Universal Robots PolyScope program: definitivo2.urp

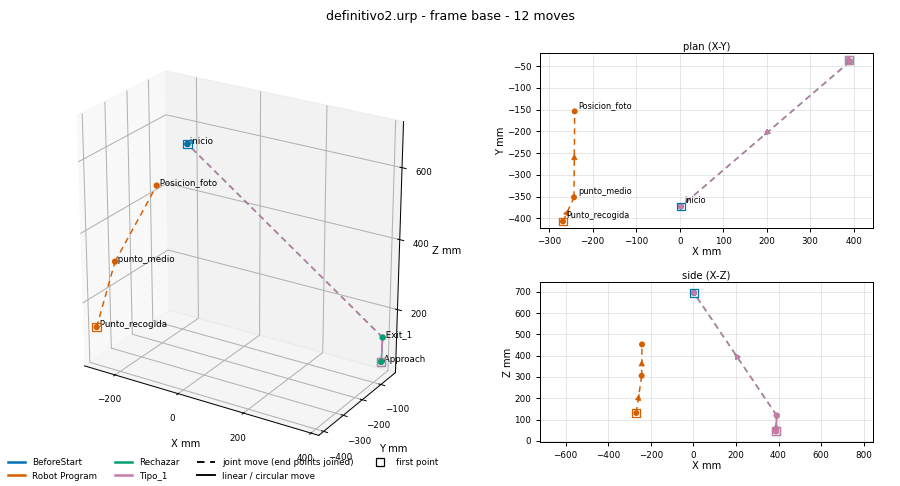
[picture p0: tool path of definitivo2.urp in frame base, 12 of 12 moves have a stored position in this frame; points joined in program order, loops and branches not executed]
Program definitivo2 (installation=default directory=/programs createdIn=5.14.5 lastSavedIn=5.14.5 robotSerialNumber=20195300809)
Calibrated DH parameters: a=[-0.000085, -0.20076, -0.212369, 0.000121, -0.000118, 0]; d=[0.15185, -26.306375, 24.753047, 1.684739, 0.085386, 0.092088]; alpha=[1.572149, -0.00522, -0.011864, 1.571339, -1.571085, 0]; deltaTheta=[0, 0.599885, -0.513355, -0.086555, 0.000006, 0]
InitVariablesNode variables(variable(name=Pallet_1_cnt_2, expression=1), variable(name=Pallet_1_cnt_3, expression=1), variable(name=Pallet_1_lct, expression=1), variable(name=Pallet_1_lct_1, expression=1), variable(name=Pallet_1_lno, expression=1), variable(name=Pallet_1_lno_1, expression=1), variable(name=Pallet_1_sep, expression=False), variable(name=Pallet_1_sep_1, expression=False), variable(name=Pallet_1_tct, expression=1), variable(name=Pallet_1_tct_1, expression=1))
BeforeStart
  MoveJ speed 60 deg/s, acceleration 80 deg/s^2 (useActiveTCP=true) feature=Base
    Waypoint inicio: TCP in base x=2.829 y=-372.735 z=694.68 mm, rx=-0.0052 ry=2.2156 rz=-2.2221 rad; joints [-0.353, -90.028, 0.079, -90.371, -0.29, 0.335] deg; TCP offset x=0 y=0 z=150 mm, rx=0 ry=0 rz=0 rad
  URCap Gripper Activate (Robotiq_Grippers, Robotiq Inc.) dataModel(ResetAndActivateKey=false)
  URCap Gripper (Robotiq_Grippers, Robotiq Inc.) dataModel(position=0.0, force=0.0, speed=100.0, positionInDouble=0.0, forceInDouble=0.0, speedInDouble=100.0, slaveIds=[3], blocking=true)
  abrir := socket_open("10.5.20.90",30003)
  Loop While (checkContinuously=false) expression=abrir≟False
    abrir := socket_open("10.5.20.90",30003)
    Wait Sleep waitTime=0.01
  vf := 0
Robot Program (runOnlyOnce=false)
  Wait Condition expression=digital_in[0]≠1
  MoveJ speed 60 deg/s, acceleration 80 deg/s^2 (useActiveTCP=true) feature=Base
    Waypoint Punto_recogida: TCP in base x=-268.281 y=-407.083 z=130.726 mm, rx=0.0255 ry=3.0678 rz=-0.0563 rad; joints [38.759, -41.295, 24.797, -71.606, -86.6, -50.187] deg
  URCap Gripper (Robotiq_Grippers, Robotiq Inc.) dataModel(position=100.0, force=100.0, speed=100.0, positionInDouble=100.0, forceInDouble=100.0, speedInDouble=100.0, slaveIds=[3], blocking=true)
  vf := 1
  MoveJ speed 60 deg/s, acceleration 80 deg/s^2 (useActiveTCP=true) feature=Base
    Waypoint punto_medio: TCP in base x=-242.896 y=-351.576 z=305.767 mm, rx=-0.0971 ry=-3.0206 rz=0.3123 rad; joints [33.768, -54.333, 0.004, -47.462, -84.671, -51.478] deg
    var_1 := 0
  df := socket_read_ascii_float(1)
  Loop While (checkContinuously=false) expression=df[1]≟0
    Wait Sleep waitTime=0.01
    df := socket_read_ascii_float(1)
  If df[1]≟1
    Call Rechazar
  ElseIf df[1]≟2
    MoveJ speed 60 deg/s, acceleration 80 deg/s^2 (useActiveTCP=true) feature=Base
      Waypoint Posicion_foto: TCP in base x=-241.348 y=-154.076 z=452.935 mm, rx=-1.8451 ry=-1.9333 rz=0.6043 rad; joints [6.803, -85.736, 5.234, -43.66, -92.516, 4.131] deg
    Script: socket_send_int(1)
    vt := socket_read_ascii_float(1)
    Loop While (checkContinuously=false) expression=vt[1]≟0
      Wait Sleep waitTime=0.01
      vt := socket_read_ascii_float(1)
    If vt≟3
      Call Tipo_1
    ElseIf vt≟4
      Call Tipo_1
    ElseIf vt≟5
      Call Tipo_1
    ElseIf vt≟6
      Call Tipo_1
    ElseIf vt≟7
      Call Rechazar
Thread Thread_2 (runOnlyOnce=false)
  Script: socket_send_line(1)
  Wait Sleep waitTime=0.01
Thread Thread_1 (runOnlyOnce=false)
  Loop While (checkContinuously=false) expression=vf≟1
    f := force()
    ff := to_str(f)
    Script: socket_send_line(ff)
    Wait Sleep waitTime=0.01
SubProgram -> Rechazar
SubProgram -> Tipo_1
SubProgram Rechazar (keepSynchronizedWithDisk=false)
  URCap Palletizing (polyscope-pallet-impl, Universal Robots) dataModel(isPalletizing=true, palletFeature=Base, Length(key=objectHeight value=0.02 unit=M), Variable(key=name, variable(name=Rechazo)), Variable(key=globalCountingVariable, variable(name=Pallet_1_cnt_2, initializeExpression=1)), Variable(key=layerCountingVariable, variable(name=Pallet_1_lct, initializeExpression=1)), Variable(key=layerNumberVariable, variable(name=Pallet_1_lno, initializeExpression=1)), Variable(key=handleSeparatorVariable, variable(name=Pallet_1_sep, initializeExpression=False)), Variable(key=totalCountVariable, variable(name=Pallet_1_tct, initializeExpression=1)), Variable(key=referencePoint, variable(featureName=referencePoint)), Variable(key=separatorPoint, variable(featureName=separatorPoint))); state(isChildrenLocked=true)
    URCap Patterns (polyscope-pallet-impl, Universal Robots) state(isChildrenLocked=true)
      URCap Pattern (polyscope-pallet-impl, Universal Robots) dataModel(UUID=9ab67c41-edff-417c-910e-e51c03855bdd, patternType=LINE, objects=3, Variable(key=nameVariable, variable(name=Line_Pattern_1))); state(isChildrenLocked=true)
        URCap Item (polyscope-pallet-impl, Universal Robots) dataModel(UUID=adfc81dc-bc46-4097-8128-33fb8ba04606, patternType=LINE, index=0, calibrationDeltaTheta=[2.0871938292282843E-8, 0.5998849625986696, -0.513354759222901, -0.08655474087847535, 6.239817607139875E-6, -6.658617090343766E-8], calibrationA=[-8.52060452638757E-5, -0.2007601879611388, -0.2123691625519033, 1.2105607098011576E-4, -1.1833705743435544E-4, 0.0], calibrationD=[0.15184970286177432, -26.306374840159272, 24.75304670983349, 1.6847390881089916, 0.085385969004481, 0.09208826337351553], calibrationAlpha=[1.5721487795181908, -0.005219907129425837, -0.011864150755780208, 1.5713392161993658, -1.5710853432049288, 0.0], calibrationJointChecksum=[-1860213401, -1859864814, -1494669377, -1328152407, -1329437658, -1329056899], calibrationStatus=2, calibrationValidChecksum=true, baseToFeature=[0.0, 0.0, 0.0, 0.0, 0.0, 0.0], TCPOffset=[-2.2911571467580313E-5, 5.575891724729498E-6, 0.15001474910538592, -3.954115798560981E-5, -6.620923200269242E-5, 1.2485531146003548E-5], JointPositions(key=jointpositions, JointPosition(key=[1], Angle(key=pos value=-0.527701 unit=RAD)), JointPosition(key=[2], Angle(key=pos value=-1.618221 unit=RAD)), JointPosition(key=[3], Angle(key=pos value=2.102014 unit=RAD)), JointPosition(key=[4], Angle(key=pos value=-2.020274 unit=RAD)), JointPosition(key=[5], Angle(key=pos value=-1.499376 unit=RAD)), JointPosition(key=[6], Angle(key=pos value=-0.528126 unit=RAD))), Variable(key=variable, variable(name=StartItem_1)))
        URCap Item (polyscope-pallet-impl, Universal Robots) dataModel(UUID=eb660494-4438-43de-8f5f-e4affd8976b3, patternType=LINE, index=1, calibrationDeltaTheta=[2.0871938292282843E-8, 0.5998849625986696, -0.513354759222901, -0.08655474087847535, 6.239817607139875E-6, -6.658617090343766E-8], calibrationA=[-8.52060452638757E-5, -0.2007601879611388, -0.2123691625519033, 1.2105607098011576E-4, -1.1833705743435544E-4, 0.0], calibrationD=[0.15184970286177432, -26.306374840159272, 24.75304670983349, 1.6847390881089916, 0.085385969004481, 0.09208826337351553], calibrationAlpha=[1.5721487795181908, -0.005219907129425837, -0.011864150755780208, 1.5713392161993658, -1.5710853432049288, 0.0], calibrationJointChecksum=[-1860213401, -1859864814, -1494669377, -1328152407, -1329437658, -1329056899], calibrationStatus=2, calibrationValidChecksum=true, baseToFeature=[0.0, 0.0, 0.0, 0.0, 0.0, 0.0], TCPOffset=[1.6778485331611116E-5, -2.1621001621285885E-6, 0.14999843934097296, -6.17118004932972E-6, 5.6336373697070044E-5, 8.147452634930435E-6], JointPositions(key=jointpositions, JointPosition(key=[1], Angle(key=pos value=-0.406319 unit=RAD)), JointPosition(key=[2], Angle(key=pos value=-1.180188 unit=RAD)), JointPosition(key=[3], Angle(key=pos value=1.651894 unit=RAD)), JointPosition(key=[4], Angle(key=pos value=-2.031068 unit=RAD)), JointPosition(key=[5], Angle(key=pos value=-1.485463 unit=RAD)), JointPosition(key=[6], Angle(key=pos value=-0.404806 unit=RAD))), Variable(key=variable, variable(name=EndItem_1)))
    URCap Layers (polyscope-pallet-impl, Universal Robots) dataModel(separators=[false], selectedPatterns=[9ab67c41-edff-417c-910e-e51c03855bdd])
    URCap At Each Item (polyscope-pallet-impl, Universal Robots) dataModel(selectedPattern=9ab67c41-edff-417c-910e-e51c03855bdd, selectedPosition=adfc81dc-bc46-4097-8128-33fb8ba04606, Approach_calibrationDeltaTheta=[2.0871938292282843E-8, 0.5998849625986696, -0.513354759222901, -0.08655474087847535, 6.239817607139875E-6, -6.658617090343766E-8], Approach_calibrationA=[-8.52060452638757E-5, -0.2007601879611388, -0.2123691625519033, 1.2105607098011576E-4, -1.1833705743435544E-4, 0.0], Approach_calibrationD=[0.15184970286177432, -26.306374840159272, 24.75304670983349, 1.6847390881089916, 0.085385969004481, 0.09208826337351553], Approach_calibrationAlpha=[1.5721487795181908, -0.005219907129425837, -0.011864150755780208, 1.5713392161993658, -1.5710853432049288, 0.0], Approach_calibrationJointChecksum=[-1860213401, -1859864814, -1494669377, -1328152407, -1329437658, -1329056899], Approach_calibrationStatus=2, Approach_calibrationValidChecksum=true, Approach_baseToFeature=[0.0, 0.0, 0.0, 0.0, 0.0, 0.0], Approach_TCPOffset=[3.3038399573775967E-6, 7.431004292735022E-6, 0.15001452865559972, -4.675145573993763E-5, -3.002590780885904E-5, 1.2382095212874822E-5], Exit_calibrationDeltaTheta=[2.0871938292282843E-8, 0.5998849625986696, -0.513354759222901, -0.08655474087847535, 6.239817607139875E-6, -6.658617090343766E-8], Exit_calibrationA=[-8.52060452638757E-5, -0.2007601879611388, -0.2123691625519033, 1.2105607098011576E-4, -1.1833705743435544E-4, 0.0], Exit_calibrationD=[0.15184970286177432, -26.306374840159272, 24.75304670983349, 1.6847390881089916, 0.085385969004481, 0.09208826337351553], Exit_calibrationAlpha=[1.5721487795181908, -0.005219907129425837, -0.011864150755780208, 1.5713392161993658, -1.5710853432049288, 0.0], Exit_calibrationJointChecksum=[-1860213401, -1859864814, -1494669377, -1328152407, -1329437658, -1329056899], Exit_calibrationStatus=2, Exit_calibrationValidChecksum=true, Exit_baseToFeature=[0.0, 0.0, 0.0, 0.0, 0.0, 0.0], Exit_TCPOffset=[-3.1032070529415923E-6, -4.811081780353721E-6, 0.14999906908731037, 3.7914955531640935E-6, -2.4690808225571853E-5, 3.2091258279986287E-6], currentWizardState=LANDING, Pose(key=refBaseToFeature, Position(key=posePosition, Length(key=X value=0 unit=M), Length(key=Y value=0 unit=M), Length(key=Z value=0 unit=M)), Rotation(key=poseRotation, Angle(key=RX value=0 unit=RAD), Angle(key=RY value=0 unit=RAD), Angle(key=RZ value=0 unit=RAD))), Pose(key=refPose, Position(key=posePosition, Length(key=X value=-0.296553 unit=M), Length(key=Y value=-0.003361 unit=M), Length(key=Z value=0.052983 unit=M)), Rotation(key=poseRotation, Angle(key=RX value=2.184884 unit=RAD), Angle(key=RY value=2.178097 unit=RAD), Angle(key=RZ value=-0.110081 unit=RAD))), JointPositions(key=Approach_jointpositions, JointPosition(key=[1], Angle(key=pos value=-0.49223 unit=RAD)), JointPosition(key=[2], Angle(key=pos value=-1.820417 unit=RAD)), JointPosition(key=[3], Angle(key=pos value=1.766277 unit=RAD)), JointPosition(key=[4], Angle(key=pos value=-1.551842 unit=RAD)), JointPosition(key=[5], Angle(key=pos value=-1.51387 unit=RAD)), JointPosition(key=[6], Angle(key=pos value=-0.434112 unit=RAD))), JointPositions(key=Exit_jointpositions, JointPosition(key=[1], Angle(key=pos value=-0.525829 unit=RAD)), JointPosition(key=[2], Angle(key=pos value=-1.798975 unit=RAD)), JointPosition(key=[3], Angle(key=pos value=1.760376 unit=RAD)), JointPosition(key=[4], Angle(key=pos value=-1.505272 unit=RAD)), JointPosition(key=[5], Angle(key=pos value=-1.420837 unit=RAD)), JointPosition(key=[6], Angle(key=pos value=-0.493217 unit=RAD))))
      URCap Generated Movements (polyscope-pallet-impl, Universal Robots) state(isChildrenLocked=true)
        MoveJ speed 60 deg/s, acceleration 80 deg/s^2 (useActiveTCP=true) feature=referencePoint
          Waypoint Approach: TCP in base x=388.088 y=-36.916 z=45.314 mm, rx=2.1976 ry=-2.1944 rz=-0.0704 rad; joints [155.436, -65.779, 88.896, -110.001, -91.77, -24.774] deg; feature pose in base x=-296.553 y=-3.361 z=52.983 mm, rx=2.1849 ry=2.1781 rz=-0.1101 rad
        MoveL speed 250 mm/s, acceleration 1200 mm/s^2 (useActiveTCP=true) feature(featureName=referencePoint)
          Waypoint ToolActionPoint: TCP in base x=388.074 y=-36.904 z=45.294 mm, rx=2.1976 ry=-2.1944 rz=-0.0705 rad; joints [155.436, -65.778, 88.898, -110.001, -91.77, -24.775] deg
        Folder Tool action
          URCap Gripper (Robotiq_Grippers, Robotiq Inc.) dataModel(position=0.0, force=10.0, speed=100.0, positionInDouble=0.0, forceInDouble=10.0, speedInDouble=100.0, slaveIds=[3], blocking=true)
        MoveL speed 250 mm/s, acceleration 1200 mm/s^2 (useActiveTCP=true) feature(featureName=referencePoint)
          Waypoint Exit_1: TCP in base x=391.496 y=-39.172 z=118.676 mm, rx=2.2265 ry=-2.2036 rz=-0.0167 rad; joints [154.845, -71.579, 77.658, -95.349, -91.108, -25.717] deg
  MoveJ speed 60 deg/s, acceleration 80 deg/s^2 (useActiveTCP=true) feature=Base
    Waypoint inicio: TCP in base x=2.829 y=-372.735 z=694.68 mm, rx=-0.0052 ry=2.2156 rz=-2.2221 rad; joints [-0.353, -90.028, 0.079, -90.371, -0.29, 0.335] deg
SubProgram Tipo_1 (keepSynchronizedWithDisk=false)
  URCap Palletizing (polyscope-pallet-impl, Universal Robots) dataModel(isPalletizing=true, palletFeature=Base, Length(key=objectHeight value=0.02 unit=M), Variable(key=name, variable(name=Rechazo_1)), Variable(key=globalCountingVariable, variable(name=Pallet_1_cnt_3, initializeExpression=1)), Variable(key=layerCountingVariable, variable(name=Pallet_1_lct_1, initializeExpression=1)), Variable(key=layerNumberVariable, variable(name=Pallet_1_lno_1, initializeExpression=1)), Variable(key=handleSeparatorVariable, variable(name=Pallet_1_sep_1, initializeExpression=False)), Variable(key=totalCountVariable, variable(name=Pallet_1_tct_1, initializeExpression=1)), Variable(key=referencePoint, variable(featureName=referencePoin_1)), Variable(key=separatorPoint, variable(featureName=separatorPoin_1))); state(isChildrenLocked=true)
    URCap Patterns (polyscope-pallet-impl, Universal Robots) state(isChildrenLocked=true)
      URCap Pattern (polyscope-pallet-impl, Universal Robots) dataModel(UUID=9ab67c41-edff-417c-910e-e51c03855bdd, patternType=LINE, objects=3, Variable(key=nameVariable, variable(name=Line_Pattern_2))); state(isChildrenLocked=true)
        URCap Item (polyscope-pallet-impl, Universal Robots) dataModel(UUID=adfc81dc-bc46-4097-8128-33fb8ba04606, patternType=LINE, index=0, calibrationDeltaTheta=[2.0871938292282843E-8, 0.5998849625986696, -0.513354759222901, -0.08655474087847535, 6.239817607139875E-6, -6.658617090343766E-8], calibrationA=[-8.52060452638757E-5, -0.2007601879611388, -0.2123691625519033, 1.2105607098011576E-4, -1.1833705743435544E-4, 0.0], calibrationD=[0.15184970286177432, -26.306374840159272, 24.75304670983349, 1.6847390881089916, 0.085385969004481, 0.09208826337351553], calibrationAlpha=[1.5721487795181908, -0.005219907129425837, -0.011864150755780208, 1.5713392161993658, -1.5710853432049288, 0.0], calibrationJointChecksum=[-1860213401, -1859864814, -1494669377, -1328152407, -1329437658, -1329056899], calibrationStatus=2, calibrationValidChecksum=true, baseToFeature=[0.0, 0.0, 0.0, 0.0, 0.0, 0.0], TCPOffset=[7.269808079073126E-6, -4.117585323482054E-6, 0.14998916095553622, 4.0003786188688346E-5, 1.3858066419453344E-5, 7.679169984422718E-5], Variable(key=variable, variable(name=StartItem_2)), JointPositions(key=jointpositions, JointPosition(key=[1], Angle(key=pos value=2.746125 unit=RAD)), JointPosition(key=[2], Angle(key=pos value=-1.145143 unit=RAD)), JointPosition(key=[3], Angle(key=pos value=1.553975 unit=RAD)), JointPosition(key=[4], Angle(key=pos value=-1.865462 unit=RAD)), JointPosition(key=[5], Angle(key=pos value=-1.654934 unit=RAD)), JointPosition(key=[6], Angle(key=pos value=-0.403705 unit=RAD))))
        URCap Item (polyscope-pallet-impl, Universal Robots) dataModel(UUID=eb660494-4438-43de-8f5f-e4affd8976b3, patternType=LINE, index=1, calibrationDeltaTheta=[2.0871938292282843E-8, 0.5998849625986696, -0.513354759222901, -0.08655474087847535, 6.239817607139875E-6, -6.658617090343766E-8], calibrationA=[-8.52060452638757E-5, -0.2007601879611388, -0.2123691625519033, 1.2105607098011576E-4, -1.1833705743435544E-4, 0.0], calibrationD=[0.15184970286177432, -26.306374840159272, 24.75304670983349, 1.6847390881089916, 0.085385969004481, 0.09208826337351553], calibrationAlpha=[1.5721487795181908, -0.005219907129425837, -0.011864150755780208, 1.5713392161993658, -1.5710853432049288, 0.0], calibrationJointChecksum=[-1860213401, -1859864814, -1494669377, -1328152407, -1329437658, -1329056899], calibrationStatus=2, calibrationValidChecksum=true, baseToFeature=[0.0, 0.0, 0.0, 0.0, 0.0, 0.0], TCPOffset=[-3.256181443245937E-5, -7.197142979531446E-6, 0.14998318903616092, 3.359344740163751E-5, -3.2320960090603836E-5, -3.9107678567338966E-5], Variable(key=variable, variable(name=EndItem_2)), JointPositions(key=jointpositions, JointPosition(key=[1], Angle(key=pos value=2.807379 unit=RAD)), JointPosition(key=[2], Angle(key=pos value=-0.748649 unit=RAD)), JointPosition(key=[3], Angle(key=pos value=0.91089 unit=RAD)), JointPosition(key=[4], Angle(key=pos value=-1.753836 unit=RAD)), JointPosition(key=[5], Angle(key=pos value=-1.603484 unit=RAD)), JointPosition(key=[6], Angle(key=pos value=-0.340183 unit=RAD))))
    URCap Layers (polyscope-pallet-impl, Universal Robots) dataModel(separators=[false], selectedPatterns=[9ab67c41-edff-417c-910e-e51c03855bdd])
    URCap At Each Item (polyscope-pallet-impl, Universal Robots) dataModel(selectedPattern=9ab67c41-edff-417c-910e-e51c03855bdd, selectedPosition=adfc81dc-bc46-4097-8128-33fb8ba04606, Approach_calibrationDeltaTheta=[2.0871938292282843E-8, 0.5998849625986696, -0.513354759222901, -0.08655474087847535, 6.239817607139875E-6, -6.658617090343766E-8], Approach_calibrationA=[-8.52060452638757E-5, -0.2007601879611388, -0.2123691625519033, 1.2105607098011576E-4, -1.1833705743435544E-4, 0.0], Approach_calibrationD=[0.15184970286177432, -26.306374840159272, 24.75304670983349, 1.6847390881089916, 0.085385969004481, 0.09208826337351553], Approach_calibrationAlpha=[1.5721487795181908, -0.005219907129425837, -0.011864150755780208, 1.5713392161993658, -1.5710853432049288, 0.0], Approach_calibrationJointChecksum=[-1860213401, -1859864814, -1494669377, -1328152407, -1329437658, -1329056899], Approach_calibrationStatus=2, Approach_calibrationValidChecksum=true, Approach_baseToFeature=[0.0, 0.0, 0.0, 0.0, 0.0, 0.0], Approach_TCPOffset=[3.3038399573775967E-6, 7.431004292735022E-6, 0.15001452865559972, -4.675145573993763E-5, -3.002590780885904E-5, 1.2382095212874822E-5], Exit_calibrationDeltaTheta=[2.0871938292282843E-8, 0.5998849625986696, -0.513354759222901, -0.08655474087847535, 6.239817607139875E-6, -6.658617090343766E-8], Exit_calibrationA=[-8.52060452638757E-5, -0.2007601879611388, -0.2123691625519033, 1.2105607098011576E-4, -1.1833705743435544E-4, 0.0], Exit_calibrationD=[0.15184970286177432, -26.306374840159272, 24.75304670983349, 1.6847390881089916, 0.085385969004481, 0.09208826337351553], Exit_calibrationAlpha=[1.5721487795181908, -0.005219907129425837, -0.011864150755780208, 1.5713392161993658, -1.5710853432049288, 0.0], Exit_calibrationJointChecksum=[-1860213401, -1859864814, -1494669377, -1328152407, -1329437658, -1329056899], Exit_calibrationStatus=2, Exit_calibrationValidChecksum=true, Exit_baseToFeature=[0.0, 0.0, 0.0, 0.0, 0.0, 0.0], Exit_TCPOffset=[-3.1032070529415923E-6, -4.811081780353721E-6, 0.14999906908731037, 3.7914955531640935E-6, -2.4690808225571853E-5, 3.2091258279986287E-6], currentWizardState=LANDING, Pose(key=refBaseToFeature, Position(key=posePosition, Length(key=X value=0 unit=M), Length(key=Y value=0 unit=M), Length(key=Z value=0 unit=M)), Rotation(key=poseRotation, Angle(key=RX value=0 unit=RAD), Angle(key=RY value=0 unit=RAD), Angle(key=RZ value=0 unit=RAD))), Pose(key=refPose, Position(key=posePosition, Length(key=X value=-0.296553 unit=M), Length(key=Y value=-0.003361 unit=M), Length(key=Z value=0.052983 unit=M)), Rotation(key=poseRotation, Angle(key=RX value=2.184884 unit=RAD), Angle(key=RY value=2.178097 unit=RAD), Angle(key=RZ value=-0.110081 unit=RAD))), JointPositions(key=Approach_jointpositions, JointPosition(key=[1], Angle(key=pos value=-0.49223 unit=RAD)), JointPosition(key=[2], Angle(key=pos value=-1.820417 unit=RAD)), JointPosition(key=[3], Angle(key=pos value=1.766277 unit=RAD)), JointPosition(key=[4], Angle(key=pos value=-1.551842 unit=RAD)), JointPosition(key=[5], Angle(key=pos value=-1.51387 unit=RAD)), JointPosition(key=[6], Angle(key=pos value=-0.434112 unit=RAD))), JointPositions(key=Exit_jointpositions, JointPosition(key=[1], Angle(key=pos value=-0.525829 unit=RAD)), JointPosition(key=[2], Angle(key=pos value=-1.798975 unit=RAD)), JointPosition(key=[3], Angle(key=pos value=1.760376 unit=RAD)), JointPosition(key=[4], Angle(key=pos value=-1.505272 unit=RAD)), JointPosition(key=[5], Angle(key=pos value=-1.420837 unit=RAD)), JointPosition(key=[6], Angle(key=pos value=-0.493217 unit=RAD))))
      URCap Generated Movements (polyscope-pallet-impl, Universal Robots) state(isChildrenLocked=true)
        MoveJ speed 60 deg/s, acceleration 80 deg/s^2 (useActiveTCP=true) feature=referencePoin_1
          Waypoint Approach: TCP in base x=388.088 y=-36.916 z=45.314 mm, rx=2.1976 ry=-2.1944 rz=-0.0704 rad; joints [155.436, -65.779, 88.896, -110.001, -91.77, -24.774] deg; feature pose in base x=-296.553 y=-3.361 z=52.983 mm, rx=2.1849 ry=2.1781 rz=-0.1101 rad
        MoveL speed 250 mm/s, acceleration 1200 mm/s^2 (useActiveTCP=true) feature(featureName=referencePoin_1)
          Waypoint ToolActionPoint: TCP in base x=388.074 y=-36.904 z=45.294 mm, rx=2.1976 ry=-2.1944 rz=-0.0705 rad; joints [155.436, -65.778, 88.898, -110.001, -91.77, -24.775] deg
        Folder Tool action
          URCap Gripper (Robotiq_Grippers, Robotiq Inc.) dataModel(position=0.0, force=10.0, speed=100.0, positionInDouble=0.0, forceInDouble=10.0, speedInDouble=100.0, slaveIds=[3], blocking=true)
        MoveL speed 250 mm/s, acceleration 1200 mm/s^2 (useActiveTCP=true) feature(featureName=referencePoin_1)
          Waypoint Exit_1: TCP in base x=391.496 y=-39.172 z=118.676 mm, rx=2.2265 ry=-2.2036 rz=-0.0167 rad; joints [154.845, -71.579, 77.658, -95.349, -91.108, -25.717] deg
  MoveJ speed 60 deg/s, acceleration 80 deg/s^2 (useActiveTCP=true) feature=Base
    Waypoint inicio: TCP in base x=2.829 y=-372.735 z=694.68 mm, rx=-0.0052 ry=2.2156 rz=-2.2221 rad; joints [-0.353, -90.028, 0.079, -90.371, -0.29, 0.335] deg
